{attribute addProperty BoxType "EK1960-2600-0019"}
{attribute addProperty Id "FSOEAT %Q*FSOE_340991D312015"}
{attribute addProperty CRC "3899632342"}
{attribute addProperty SizeInBites "120"}
{attribute addProperty SizeInBytes "15"}
TYPE FSoE_Outputs_E86FAAD6 :
STRUCT
	{attribute addProperty Name "FSOE"}
	FSOE AT %Q* : FSOE_340991D3;
END_STRUCT
END_TYPE

(* stored: Version 1.2.0.0, ProductVersion 3.1.4024.9
   DUT FSoE_Outputs_E86FAAD6: Id {5e53d85d-da64-4dec-a673-6ee2e5a878ef} *)
